FUNCTION_BLOCK Vision_Inspection_HMI EXTENDS StateControllerHMI
VAR
END_VAR

PROPERTY ControlObject : I_Base
SET
END_SET
END_PROPERTY

METHOD CyclicLogic
VAR_INST
	StartRT : R_TRIG;
	StopRT	: R_TRIG;
	ResetRT : R_TRIG;
END_VAR
SUPER^.CyclicLogic();

// User buttons
Statemachine_HMI.StartPermissive := Statemachine_HMI.CurrentState = E_PMLState.Idle;
Statemachine_HMI.StopPermissive	 := Statemachine_HMI.CurrentState <> E_PMLState.Aborted;
Statemachine_HMI.ResetPermissive := Statemachine_HMI.CurrentState = E_PMLState.Aborted OR Statemachine_HMI.CurrentState = E_PMLState.Stopped;
StartRT(CLK := Statemachine_HMI.StartPressed);
IF StartRT.Q THEN
	_stateMachine.RequestStart();
END_IF

StopRT(CLK := Statemachine_HMI.StopPressed);
IF StopRT.Q THEN
	IF Statemachine_HMI.CurrentState = E_PMLState.Stopped THEN
		_stateMachine.RequestAbort();
	ELSE
		_stateMachine.RequestStop();
	END_IF
END_IF

ResetRT(CLK := Statemachine_HMI.ResetPressed);
IF ResetRT.Q THEN
	IF Statemachine_HMI.CurrentState = E_PMLState.Aborted THEN
		_stateMachine.RequestClear();
	ELSE
		_stateMachine.RequestReset();
	END_IF
END_IF
END_METHOD

END_FUNCTION_BLOCK

(* stored: Version 1.1.0.1
   POU Vision_Inspection_HMI: Id {d1d46972-f2fd-4223-8233-5df0f2317bba}, SpecialFunc None
   Property ControlObject: Id {b19ed197-897a-4f85-98a2-f1a3519f7b04}
   Set Set: Id {e7384cab-71c7-4c4d-9342-664ea9234160}
   Method CyclicLogic: Id {31cd966e-8062-4cc6-89e1-b6a373b81562} *)
